TYPE "IAI Par Struct"
VERSION : 0.1
   STRUCT
      AxisID : Int;
      PositionWidth : Real;
      PosCode : Int;
      PushDir : Int;
      PushWidth : Real;
      PushCurrent : Int;
      TargetPosition : Array[0..49] of Real;
      GoPosInterfere : Array[0..99] of Bool;
      Speed : Int;
      Acceleration : Int;
      ChgSpeed : Int;
      PushSpeed : Int;
      WritePosition : Real;
      AlarmTime : Time;
   END_STRUCT;

END_TYPE

